ABB RAPID module: program.mod

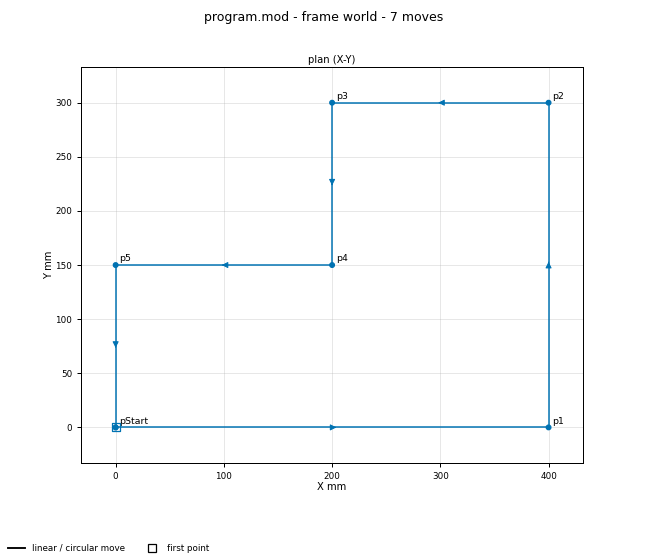
[picture p0: tool path of program.mod in frame world, 7 of 7 moves have a stored position in this frame; points joined in program order, loops and branches not executed]
MODULE TrajectorySim
    ! ==========================================
    ! Generated by Python Trajectory Simulator
    ! https://github.com/tuousername/robot-trajectory-sim
    ! ==========================================
    CONST robtarget pStart := [[0.0, 0.0, 0.0], [1, 0, 0, 0], [0, 0, 0, 0], [9E9, 9E9, 9E9, 9E9, 9E9, 9E9]];

    CONST robtarget p1 := [[400.0, 0.0, 0.0], [1, 0, 0, 0], [0, 0, 0, 0], [9E9, 9E9, 9E9, 9E9, 9E9, 9E9]];
    CONST robtarget p2 := [[400.0, 300.0, 0.0], [1, 0, 0, 0], [0, 0, 0, 0], [9E9, 9E9, 9E9, 9E9, 9E9, 9E9]];
    CONST robtarget p3 := [[200.0, 300.0, 0.0], [1, 0, 0, 0], [0, 0, 0, 0], [9E9, 9E9, 9E9, 9E9, 9E9, 9E9]];
    CONST robtarget p4 := [[200.0, 150.0, 0.0], [1, 0, 0, 0], [0, 0, 0, 0], [9E9, 9E9, 9E9, 9E9, 9E9, 9E9]];
    CONST robtarget p5 := [[0.0, 150.0, 0.0], [1, 0, 0, 0], [0, 0, 0, 0], [9E9, 9E9, 9E9, 9E9, 9E9, 9E9]];
    CONST robtarget p6 := [[0.0, 0.0, 0.0], [1, 0, 0, 0], [0, 0, 0, 0], [9E9, 9E9, 9E9, 9E9, 9E9, 9E9]];

    PROC main()
        ! Move to start position
        MoveL pStart, v100, fine, weldGun1;

        ! Segment 1: speed=150mm/s, zone=z5
        MoveL p1, v150, z5, weldGun1;

        ! Segment 2: speed=80mm/s, zone=z1
        MoveL p2, v80, z1, weldGun1;

        ! Segment 3: speed=100mm/s, zone=z5
        MoveL p3, v100, z5, weldGun1;

        ! Segment 4: speed=60mm/s, zone=z0
        MoveL p4, v60, z0, weldGun1;

        ! Segment 5: speed=100mm/s, zone=z5
        MoveL p5, v100, z5, weldGun1;

        ! Segment 6: speed=120mm/s, zone=fine
        MoveL p6, v120, fine, weldGun1;

    ENDPROC
ENDMODULE
